{attribute 'strict'}
TYPE E_FileLoggerSetNewPathState :
(
	FILE_LOGGER_SET_NEW_PATH_CHANGE_PATH			:= 0,
	FILE_LOGGER_SET_NEW_PATH_DONE					:= 10
);
END_TYPE

(* stored: Version 1.1.0.1, ProductVersion 3.1.4024.9
   DUT E_FileLoggerSetNewPathState: Id {9f1f4044-0810-4eb2-a537-81f18142ddfa} *)
